Yaskawa INFORM job: R1_W72(-45,-90)KM-OK.JBI

/JOB
//NAME R1_W72(-45,-90)KM-OK
///FOLDERNAME KRIS-SCIANA
//POS
///NPOS 54,54,0,3,0,0
///TOOL 0
///POSTYPE PULSE
///PULSE
C00000=22665,120049,18248,-11675,101032,82300
C00001=-122130,43329,-6683,12152,111441,19153
C00002=-120622,72164,45661,10422,113266,19720
C00003=-120624,72162,45658,10422,113267,19719
C00004=-120625,70696,44450,10437,113255,19718
C00005=-120625,69731,43760,10431,113184,19712
C00006=-120625,72161,45657,10422,113267,19719
C00007=-120625,73217,47541,-436,111867,18871
C00008=-120625,75029,50702,-434,110853,18873
C00009=-120625,72176,45675,-438,112481,18869
C00010=-120625,72178,45676,-438,112481,18869
C00011=-120622,72181,45681,-437,112480,18870
C00012=-120616,72075,45554,-489,94840,46442
C00013=-120618,72071,45549,-489,94840,46441
C00014=-120642,73345,48177,-487,93880,46436
C00015=-120642,72353,47400,-487,93849,46436
C00016=-120642,73345,48177,-487,93880,46436
C00017=-120642,74197,49572,-487,93477,46436
C00018=-120619,72071,45549,-489,94840,46441
C00019=-121372,78507,50594,-464,95039,46186
C00020=-120018,75037,50235,-510,93486,46650
C00021=-120417,76344,52308,-497,92881,46517
C00022=-120621,72059,44969,-489,95191,46439
C00023=-120619,72084,45565,-489,94838,46441
C00024=-120616,72075,45554,-489,94840,46442
C00025=-113201,-21187,-38102,-23980,83591,-65072
C00026=-113206,-19774,-20442,-24692,74306,-63151
C00027=-113798,-18750,-15552,-24863,71864,-62851
C00028=-114312,-17134,-12027,-24921,70492,-62748
C00029=-113978,-20043,-15729,-24898,71303,-62798
C00030=-113966,-17046,-13518,-24877,71470,-62830
C00031=-123235,-18525,-15698,-22699,69330,-65982
C00032=-133441,-17143,-17468,-19679,68369,-69735
C00033=-133995,-17029,-17893,-19478,68539,-69974
C00034=-133989,-18400,-20373,-19378,69318,-70104
C00035=-133987,-19144,-25030,-19106,71669,-70494
C00036=-133980,-18907,-41468,-18396,81392,-72016
C00037=-147817,38041,11634,3124,80895,-84927
C00038=-152519,43301,26371,4433,74738,-86715
C00039=-133823,25172,12114,-18031,70253,-81214
C00040=-133774,21924,9079,-18025,70454,-81226
C00041=-152412,43459,26540,4406,74711,-86679
C00042=-150649,40862,24360,3938,74631,-86067
C00043=-146674,34879,18639,2861,74908,-84673
C00044=-134201,24776,12665,-17966,69647,-81260
C00045=-130088,28311,21253,-29010,69005,-78746
C00046=-129790,28541,21763,-29119,68938,-78606
C00047=-129499,29238,22824,-29245,68780,-78445
C00048=-126960,34903,31839,-30366,67381,-77007
C00049=-126120,32474,24084,-29868,70737,-77592
C00050=-134008,23343,8440,-20620,71526,-80564
C00051=-134003,24203,-7351,-19847,81091,-82192
C00052=-136638,-147031,-131688,-19613,26010,-82415
C00053=-92376,-140993,-131688,-19613,26010,81348
BC00000=138740,5300,1068817
BC00001=361090,82938,964237
BC00002=361090,82938,964237
BC00003=360421,82979,937449
BC00004=360154,82996,926730
BC00005=360154,82996,926730
BC00006=360154,82996,926733
BC00007=377601,80610,926129
BC00008=377601,80610,926129
BC00009=377601,80610,926129
BC00010=378413,80544,936525
BC00011=380444,80377,962513
BC00012=252794,58026,1043699
BC00013=249819,57728,1018783
BC00014=248629,57608,1008817
BC00015=248629,57608,1008817
BC00016=248629,57608,1008817
BC00017=248629,57608,1008817
BC00018=250968,56602,1006807
BC00019=266308,55395,1001700
BC00020=266305,60542,981324
BC00021=266305,60542,981324
BC00022=266305,60542,981324
BC00023=266308,55395,1001700
BC00024=252794,58026,1043699
BC00025=398174,123466,1075175
BC00026=398174,123466,1075175
BC00027=398174,123570,1075175
BC00028=398174,123613,1075170
BC00029=398174,123612,1075175
BC00030=398174,123612,1075175
BC00031=366304,128529,1075170
BC00032=330537,134045,1075175
BC00033=330537,134045,1075175
BC00034=331080,134003,1075175
BC00035=332435,133899,1075175
BC00036=332435,133899,1075175
BC00037=322655,79873,1075174
BC00038=322653,79872,1075175
BC00039=322653,79872,1075175
BC00040=322653,79872,1075175
BC00041=322653,79872,1075175
BC00042=322653,79872,1075175
BC00043=322653,79872,1075175
BC00044=322653,79872,1075175
BC00045=336283,82967,1075175
BC00046=336283,82967,1075175
BC00047=336283,82967,1075175
BC00048=336283,82967,1075175
BC00049=336292,82968,1075175
BC00050=339912,83266,1075175
BC00051=339912,83266,1075175
BC00052=339911,83264,1075173
BC00053=155306,23208,1075173
///POSTYPE BASE
///RECTAN
///RCONF 0,0,0,0,1,0,0,0,0,0,0,0,0,0,0,0,0,0,0,0,0,0,0,0
P00006=2.006,1.622,-0.565,0.0000,0.0000,0.0000
P00021=0.073,2.058,-0.109,0.0000,0.0000,0.0000
P00022=2.006,1.622,-0.565,0.0000,0.0000,0.0000
//INST
///DATE 2024/09/12 13:36
///ATTR SC,RW
///GROUP1 RB1,BS1
NOP
'r1_W72(-45,-90)
'Path S891
SFTOF
MOVJ C00000 BC00000 VJ=100.00
MOVJ C00001 BC00001 VJ=100.00
MOVJ C00002 BC00002 VJ=100.00
MOVJ C00003 BC00003 VJ=100.00
MOVL C00004 BC00004 V=60.0
REFP 3 C00005 BC00005
CALL JOB:SEARCH-R1
SET P022 P006
SFTON P022
MOVL C00006 BC00006 V=60.0
MOVL C00007 BC00007 V=60.0
REFP 3 C00008 BC00008
CALL JOB:SEARCH-R1
SET P022 P006
SFTON P022
MOVL C00009 BC00009 V=60.0
MOVL C00010 BC00010 V=166.7
MOVL C00011 BC00011 V=166.7
'Path S1463
SFTOF
MOVJ C00012 BC00012 VJ=100.00
MOVJ C00013 BC00013 VJ=100.00
MOVL C00014 BC00014 V=60.0
REFP 3 C00015 BC00015
CALL JOB:SEARCH-R1
SET P021 P006
SFTON P021
MOVL C00016 BC00016 V=50.0
REFP 3 C00017 BC00017
CALL JOB:SEARCH-R1
SET P021 P006
SFTON P021
MOVL C00018 BC00018 V=60.0
MOVL C00019 BC00019 V=100.0
MOVL C00020 BC00020 V=60.0
REFP 3 C00021 BC00021
CALL JOB:SEARCH-R1
SET P021 P006
SFTON P021
MOVL C00022 BC00022 V=60.0
MOVL C00023 BC00023 V=100.0
MOVL C00024 BC00024 V=1000.0
'Path W19
SFTOF
SFTON P022
MOVJ C00025 BC00025 VJ=100.00
MOVJ C00026 BC00026 VJ=100.00
MOVJ C00027 BC00027 VJ=100.00
CALL JOB:COFNIJ_DRUT
MOVL C00028 BC00028 V=100.0 PL=0
REFP 1 C00029 BC00029
REFP 2 C00030 BC00030
MACRO1 MJ#(0) ARGF9
ARCON
SFTON P021
MOVL C00031 BC00031 V=10.8
MOVL C00032 BC00032 V=10.8
MOVL C00033 BC00033 V=10.8
ARCOF
MOVL C00034 BC00034 V=166.7
SFTOF
MOVL C00035 BC00035 V=166.7
MOVL C00036 BC00036 V=166.7
SFTON P021
MOVJ C00037 BC00037 VJ=50.00
MOVL C00038 BC00038 V=100.0 PL=0
REFP 1 C00039 BC00039
REFP 2 C00040 BC00040
MACRO1 MJ#(0) ARGF7
ARCON
MOVL C00041 BC00041 V=11.0
MOVL C00042 BC00042 V=10.8
MOVL C00043 BC00043 V=10.8
MOVL C00044 BC00044 V=10.8
MOVL C00045 BC00045 V=10.8
MOVL C00046 BC00046 V=10.8
MOVL C00047 BC00047 V=10.8
MOVL C00048 BC00048 V=10.8
ARCOF
MOVL C00049 BC00049 V=166.7
MOVL C00050 BC00050 V=166.7
MOVL C00051 BC00051 V=166.7
SFTOF
MOVJ C00052 BC00052 VJ=100.00
MOVJ C00053 BC00053 VJ=100.00
END
